INTERFACE I_TemperatureSensor

PROPERTY Temperature : REAL
GET
END_GET
END_PROPERTY

END_INTERFACE

(* stored: Version 1.1.0.1
   Itf I_TemperatureSensor: Id {83bb4304-a51b-4ad9-a3b6-6fe0a375e02b}
   Property Temperature: Id {79d7e23f-7f45-45e3-9b0f-3b9a5ace9663}
   Get Get: Id {bc210361-8fe6-461a-bdc7-2546ec0f0903} *)
